FUNCTION_BLOCK Safety_Hmi
VAR_GENERIC CONSTANT
	ESTOP_CAP		: UDINT := 4;
END_VAR

VAR_INPUT
	bEStopActive	: ARRAY[1..ESTOP_CAP] OF BOOL;
	
	sStatusText		: Str;
	nStatusColor	: Color;
	
	bReset			: BOOL;
	bHideReset		: BOOL;
END_VAR

END_FUNCTION_BLOCK

(* stored: Version 1.1.0.1
   POU Safety_Hmi: Id {4d75a0c5-3298-465d-849c-fb6bf543b76a}, SpecialFunc None *)
